FUNCTION_BLOCK SKILL_Release (* Releases the equipment a module level skill holds after a failure or abort: (Token, safe command 0, release) for the equipment command channels *)
  (* Standard: 61499-2 *)
  (* Version 0.1, 2026-09-28, Project contributors, AAU Smart Production Lab *)
  PACKAGE modlib;
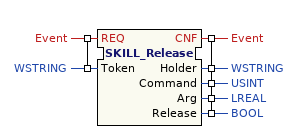
  EVENT_INPUT
    REQ WITH Token;
  END_EVENT
  EVENT_OUTPUT
    CNF WITH Holder, Command, Arg, Release;
  END_EVENT
  VAR_INPUT
    Token : WSTRING;
  END_VAR
  VAR_OUTPUT
    Holder : WSTRING;
    Command : USINT;
    Arg : LREAL;
    Release : BOOL;
  END_VAR
  EC_STATES
    REQ : REQ -> CNF;
  END_STATES
  ALGORITHM REQ IN ST:
Holder := Token;
Command := 0;
Arg := 0.0;
Release := TRUE;
  END_ALGORITHM
END_FUNCTION_BLOCK
